PROGRAM P_Demo_F_BA_CheckEnum
VAR
    argNIndex                      : INT                            := 0; // nIndex
    ioAInfo                        : ARRAY [*] OF ST_BA_EnumInfo; // aInfo 双向
    fnReturn                       : BOOL; // 返回值
END_VAR

// =============================================================================
// Tc3_BA2_Common.F_BA_CheckEnum 演示程序
// =============================================================================
// 场景：运行时检查 HMI 传入的枚举值合法性："用户选择的传感器类型代码是否在我支持的列表里"。
//
// 价值：一行 FC 替代手写 FOR 循环遍历查找。
//
// 验证：登录 PLC 后，按例程内变量在线写值；监视输出 / 返回值，结合 §1 功能
//       简述的预期行为对照（详见配套 .md 文档 §7 业务场景）。
//
// 验证步骤：
//   1. 右键 PLC 项目下 POUs 文件夹 → Add → Existing Item → 选本 .TcPOU 文件
//   2. 引用 Tc3_BA2_Common（References → Add library）
//   3. 编译 → 登录 → 运行；按上方『验证』指引在线写值观察
// =============================================================================

fnReturn := F_BA_CheckEnum(
    nIndex                   := argNIndex,
    aInfo                    := ioAInfo
);

END_PROGRAM

(* stored: Version 1.1.0.1, ProductVersion 3.1.4024.5
   POU P_Demo_F_BA_CheckEnum: Id {56c50859-ebb6-53ec-a60c-054c1379eb2e}, SpecialFunc None *)
